SUBAPPLICATION Button_CLIENT_Method_IE (* VT-Button (Button_IE) loest per CLIENT_0 einen entfernten argument- und rueckgabewertlosen OPC-UA-Methodenaufruf (ACTION=CALL_METHOD) aus - allgemeines Muster fuer 'VT-Taste ruft eine Methode auf einer anderen Station auf', herausgeloest aus logiBUS_AI_Calibrated_Subscribe_VT_OPC (CO/CS kamen dort 2x identisch vor, siehe OPC_UA_VERNETZUNG.md Punkt 14). Analog zu Button_Method_IE (dort: Button ODER lokale Methode -> gemeinsames IND), hier aber der umgekehrte 'Caller'-Fall: Button -> entfernte Methode. *)
  (* Standard: 61499-2; Description: Copyright (c) 2026 Meisterschulen am Ostbahnhof This program and the accompanying materials are made available under the terms of the Eclipse Public License 2.0 which is available at https://www.eclipse.org/legal/epl-2.0/ SPDX-License-Identifier: EPL-2.0 *)
  (* Version 1.0, 2026-09-22, Franz Höpfinger, Meisterschulen am Ostbahnhof, initial implementation - herausgeloest aus logiBUS_AI_Calibrated_Subscribe_VT_OPC (Button_IE + CLIENT_0 kam dort 2x identisch vor, fuer CO und CS). Franz: 'Button_IE CLIENT_0 kann eine Subapp werden, das ist ein generelles Muster zum Rufen einer Methode vom VT aus' - InputEvent ist Parameter (nicht hartcodiert auf BT_PRESSED_LATCHED), damit auch andere Aktivierungsarten (z.B. Loslassen) wiederverwendbar sind. *)
  PACKAGE MyLib::sys;
  IMPORT isobus::UT::io::Button::ButtonActivationCode_S;
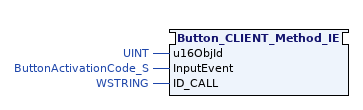
  VAR_INPUT
    u16ObjId : UINT; (* Object ID Button *)
    InputEvent : isobus::UT::io::Button::ButtonActivationCode_S; (* Welche Button-Aktivierung den Methodenaufruf ausloest (z.B. BT_PRESSED_LATCHED, BT_RELEASED_UNLATCHED) *)
    ID_CALL : WSTRING; (* Remote-Methodenadresse (ACTION=CALL_METHOD) - ruft die entsprechende ID_..._METHOD-Adresse (ACTION=CREATE_METHOD) auf der Zielstation auf *)
  END_VAR
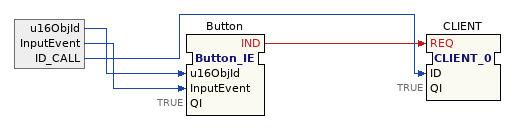
  FBS
    Button : isobus::UT::io::Button::Button_IE(QI := TRUE);
    CLIENT : iec61499::net::CLIENT_0(QI := TRUE);
  END_FBS
  EVENT_CONNECTIONS
    Button.IND TO CLIENT.REQ;
  END_CONNECTIONS
  DATA_CONNECTIONS
    u16ObjId TO Button.u16ObjId;
    InputEvent TO Button.InputEvent;
    ID_CALL TO CLIENT.ID;
  END_CONNECTIONS
END_SUBAPPLICATION
